FUNCTION_BLOCK bk5xxxBasicAxis_FB EXTENDS BeckHoffBasicAxis_FB
VAR_INPUT
	pDigIn: 	POINTER TO INT;	
END_VAR
VAR_OUTPUT
END_VAR
VAR
	
END_VAR


AxisCtrlPtr^.Input.Parameter.Drive.eDriveType	:= enumDriveType.e5xxxBeckhoff;
AxisCtrlPtr^.Input.Parameter.Drive.VendorNameID	:= eVendorNameID.Beckhoff;


SUPER^(AxisRef:=AxisRef);

IF (pDigIn <> 0) THEN
	AxisCtrlPtr^.Output.Status.DriveEnable	:= pDigIn^.7;
ELSE
	AxisCtrlPtr^.Output.Status.DriveEnable	:= TRUE;
END_IF

END_FUNCTION_BLOCK

(* stored: Version 1.1.0.1, ProductVersion 3.1.4024.3
   POU bk5xxxBasicAxis_FB: Id {b77b2bc0-2247-4c7a-bd38-3884568fedd8}, SpecialFunc None *)
